Fanuc KAREL source: kc00025.KL

-- PROVISIONAL review KL for V770-1; original PC SHA256 465325bae714bea94a45ae1fd8aff74d4c25fcb40761f55c0421cfe511eff661
-- Incomplete behavior may be omitted. Consult companion uncertainty JSON. Do not deploy.
PROGRAM KC00025
%NOLOCKGROUP
BEGIN
  -- UNRESOLVED_PC offsets 5-17; opcodes 3F,75
  -- UNRESOLVED_PC offsets 22-64; opcodes 27,22,2A,22,22,22,22,22,31
  -- UNRESOLVED_PC offsets 69-73; opcodes 7F
END KC00025
